{attribute 'no_explicit_call' := 'This FB is a CLASS and must be accessed using methods or properties'}
FUNCTION_BLOCK FB_DrawAxis EXTENDS FB_PackML_BaseModule
VAR
	Axis	  : FB_Component_BasicSlaveAxis := (Name := 'Draw Axis');
	MasterRef : REFERENCE TO AXIS_REF;
END_VAR

METHOD PROTECTED Aborting
// Mode is ignored
CASE SequenceState OF
	0:
		NoStateTasksToComplete := FALSE;
		SequenceState		   := SequenceState + 10;

	10: // Stop Axis
		Axis.Override := 100;
		Axis.Stop(); // This will also GearOut by default
		IF Axis.Stopped THEN
			SequenceState := SequenceState + 10;
		END_IF

	20: // Disable Axis
		Axis.Disable();
		IF NOT Axis.Enabled THEN
			StateTasksComplete := TRUE;
		END_IF
END_CASE

SUPER^.Aborting();
END_METHOD

PROPERTY AxisRef : REFERENCE TO AXIS_REF
GET
AxisRef REF= Axis.Axis;
END_GET
END_PROPERTY

METHOD PROTECTED Completing
CASE _CurrentMode OF
	ePMLUnitMode_Production:
		CASE SequenceState OF
			0:
				NoStateTasksToComplete := FALSE;
				SequenceState		   := SequenceState + 10;

			10: // Wait for Master Axis to Stop and GearOut, or Stop
				IF Axis.InGear AND Axis.Stopped THEN
					Axis.GearOut();
				ELSIF NOT Axis.InGear THEN
					Axis.Stop();
				END_IF

				IF Axis.Stopped THEN
					StateTasksComplete := TRUE;
				END_IF
		END_CASE
END_CASE

SUPER^.Completing();
END_METHOD

METHOD PUBLIC CyclicLogic
IF NOT _InitComplete THEN
	_InitComplete := Initialize();
	RETURN;
END_IF

SUPER^.CyclicLogic();
END_METHOD

METHOD PROTECTED Initialize : BOOL;
VAR
	i : UDINT;
END_VAR
Initialize := FALSE;
CASE DescendantSequenceState OF
	0: // Register Components
		RegisterComponent(Axis);

		// Set Config
		_LogModeChanges			:= FALSE;
		_LogStateChanges		:= FALSE;
		DescendantSequenceState := DescendantSequenceState + 10;

	10: // Copy Mode names
		FOR i := 1 TO 10 DO
			ModeNames[i] := F_UnitModeToString(UDINT_TO_DINT(i));
		END_FOR

		DescendantSequenceState := DescendantSequenceState + 10;

	20:
		IF SUPER^.Initialize() THEN
			DescendantSequenceState := DescendantSequenceState + 10;
		END_IF

	30:
		Initialize := TRUE;
END_CASE
END_METHOD

PROPERTY MasterAxisRef : REFERENCE TO AXIS_REF
SET
MasterRef REF= MasterAxisRef;
END_SET
END_PROPERTY

METHOD PROTECTED Starting
CASE _CommandedMode OF
	ePMLProtUnitMode_Production:
		CASE SequenceState OF
			0:
				NoStateTasksToComplete := FALSE;
				SequenceState		   := SequenceState + 10;

			10: // Enable Axis
				Axis.Enable();
				IF Axis.Enabled THEN
					SequenceState := SequenceState + 10;
				END_IF

			20: // Set reference to Master and Couple Axes
				Axis.Master1 REF= MasterRef;
				Axis.GearIn();
				IF Axis.InGear THEN
					StateTasksComplete := TRUE;
				END_IF
		END_CASE
END_CASE

SUPER^.Starting();
END_METHOD

METHOD PROTECTED Stopping
CASE _CurrentMode OF
	ePMLUnitMode_Production:
		CASE SequenceState OF
			0:
				NoStateTasksToComplete := FALSE;
				SequenceState		   := SequenceState + 10;

			10: // Stop Axis
				Axis.Override := 100;
				Axis.Stop(); // This will also GearOut by default
				IF Axis.Stopped THEN
					StateTasksComplete := TRUE;
				END_IF
		END_CASE
END_CASE

SUPER^.Stopping();
END_METHOD

END_FUNCTION_BLOCK

(* stored: Version 1.1.0.1, ProductVersion 3.1.4024.12
   POU FB_DrawAxis: Id {6f7f3fdd-1761-46b2-a834-6c3784a9206a}, SpecialFunc None
   Folder Methods: Id {1459c28b-8a12-4641-8a5e-d74da0b71b0d}
   Folder Properties: Id {2a6d81ec-4259-4ac1-afbc-17e71288b5f6}
   Method Aborting: Id {d947f5e2-2d16-49a5-9815-3f039233a9f0}
   Property AxisRef: Id {6a546205-aa1a-4058-a964-b861546a6b3a}
   Get Get: Id {c2ba8eac-8f12-4d77-bfd7-5fb7b5eee94d}
   Method Completing: Id {1a88739c-e241-40e6-932c-4e770d465d42}
   Method CyclicLogic: Id {071f67bd-24e9-4734-8fa9-d70acebb508f}
   Method Initialize: Id {aa1d8f3c-de5d-440d-88b2-cf20a1bca6eb}
   Property MasterAxisRef: Id {c8aeeb47-6497-45ee-b23a-b03bca698c96}
   Set Set: Id {4c5a7eeb-c2c9-4a9d-9b74-c57a2ad6979d}
   Method Starting: Id {08b85550-4819-4b11-b046-f4ec48d539b6}
   Method Stopping: Id {2444f023-ed59-4632-8f42-8076dedaa106} *)
